% RSLogix 500 project TEST_OCT_21_2019_BAK040.RSS, saved by version 11.00.00.00 %
PROJECT "UNTITLED"    % processor: MicroLogix 1200 %

PROGRAM FILES
  LAD 2   14 rungs
  LAD 3, 4, 5, 6, 7, 8, 9, 10, 11, 12, 13, 14, 15: only END

DATA FILES
  O0 OUTPUT  4 elements
  I1 INPUT  4 elements
  S2 STATUS  66 elements
  B3 BINARY  32 elements
  T4 TIMER  40 elements
  C5 COUNTER  32 elements
  R6 CONTROL  16 elements
  N7 INTEGER  105 elements
  F8 FLOAT  1 elements

LADDER 2
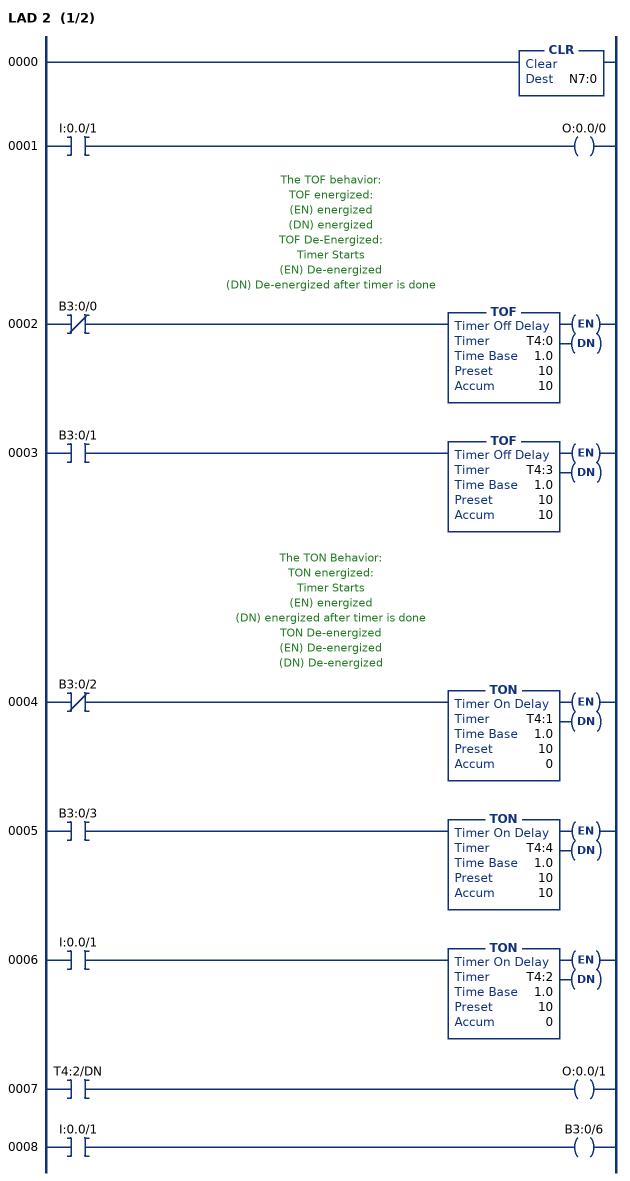
% Rung: 0 %  % edit flag set %
SOR CLR N7:0 EOR
% Rung: 1 %
SOR XIC I:0.0/1 OTE O:0.0/0 EOR
% Rung: 2 %
% The TOF behavior:
% 
% TOF energized:
% (EN) energized
% (DN) energized
% 
% TOF De-Energized:
% Timer Starts
% (EN) De-energized
% (DN) De-energized after timer is done %
SOR XIO B3:0/0 TOF T4:0 1.0 10 10 EOR
% Rung: 3 %
SOR XIC B3:0/1 TOF T4:3 1.0 10 10 EOR
% Rung: 4 %
% The TON Behavior:
% 
% TON energized:
% Timer Starts
% (EN) energized
% (DN) energized after timer is done
% 
% TON De-energized
% (EN) De-energized
% (DN) De-energized %
SOR XIO B3:0/2 TON T4:1 1.0 10 0 EOR
% Rung: 5 %
SOR XIC B3:0/3 TON T4:4 1.0 10 10 EOR
% Rung: 6 %
SOR XIC I:0.0/1 TON T4:2 1.0 10 0 EOR
% Rung: 7 %
SOR XIC T4:2/DN OTE O:0.0/1 EOR
% Rung: 8 %
SOR XIC I:0.0/1 OTE B3:0/6 EOR

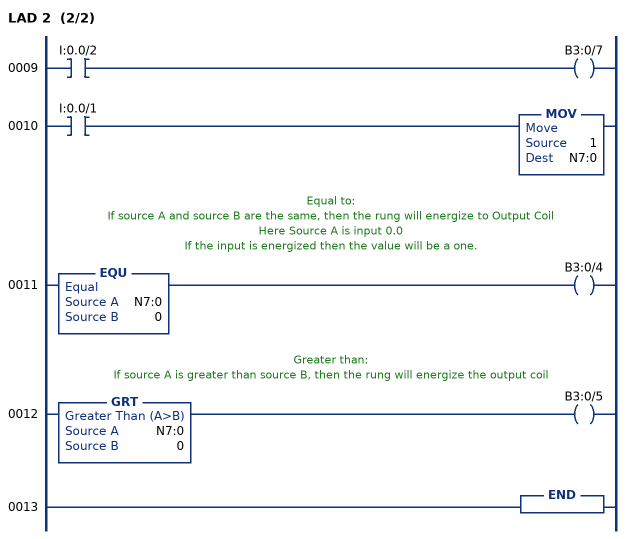
% Rung: 9 %
SOR XIC I:0.0/2 OTE B3:0/7 EOR
% Rung: 10 %
SOR XIC I:0.0/1 MOV 1 N7:0 EOR
% Rung: 11 %
% Equal to:
% 
% If source A and source B are the same, then the rung will energize to Output Coil
% 
% Here Source A is input 0.0
% If the input is energized then the value will be a one. %
SOR EQU N7:0 0 OTE B3:0/4 EOR
% Rung: 12 %
% Greater than:
% 
% If source A is greater than source B, then the rung will energize the output coil %
SOR GRT N7:0 0 OTE B3:0/5 EOR
% Rung: 13 %
SOR END EOR

DATA TABLE (non-zero values as saved)
DATA B3
% B3:0 % 0X000D 0X0000 0X0000 0X0000 0X0000 0X0000 0X0000 0X0000 0X0000 0X0000
DATA T4
% .PRE .ACC %
% T4:0 % 10 10
% T4:1 % 10 0
% T4:2 % 10 0
% T4:3 % 10 10
% T4:4 % 10 10
